// TwinCAT 3 PLC project Untitled1
// ProgramVersion: 3.1.4023.0
// libraries:
//   Tc2_Standard, * (Beckhoff Automation GmbH)
//   Tc2_System, * (Beckhoff Automation GmbH)
//   Tc2_Utilities, * (Beckhoff Automation GmbH)
//   Tc3_Database, * (Beckhoff Automation GmbH)
//   Tc3_Module, * (Beckhoff Automation GmbH)
// project tree:
//   DUTs/ ExcelInfo.TcDUT, ST_AccessConnectionInfo.TcDUT, ST_datastruct.TcDUT, st_DBInfo.TcDUT, st_InsertData.TcDUT (not stored), ST_mongoDBConnectionInfo.TcDUT, ST_MYSQLConnectionInfo.TcDUT, ST_ReturnBetweenDates.TcDUT, ST_ReturnedData_mysql_access.TcDUT, ST_SQLiteConnectionInfo.TcDUT, test.TcDUT
//   / PlcTask.TcTTO
//   POUs/ fb_ConnectDB.TcPOU, fb_CreateTable.TcPOU, fb_DBSRVCreateTable.TcPOU, fb_datareturn.TcPOU, fb_DBSRVdatareturn.TcPOU, fb_DBWrite.TcPOU, fb_DBSRVInsertRecord.TcPOU, MAIN.TcPOU

CONFIGURATION Untitled1
    RESOURCE PLC ON TwinCAT3
        TASK PlcTask(INTERVAL := T#1ms, PRIORITY := 20);
        PROGRAM MAIN WITH PlcTask : MAIN;
    END_RESOURCE
END_CONFIGURATION

// ---- DUTs/ExcelInfo.TcDUT
TYPE ExcelInfo :
STRUCT
	ColumnName:STRING(50):='';
	ColumnNumber:INT:=0;
	bready:BOOL:=FALSE;
	path:STRING(200):='';
END_STRUCT
END_TYPE

// ---- DUTs/ST_AccessConnectionInfo.TcDUT
TYPE ST_AccessConnectionInfo :
STRUCT
	Path:STRING(255);
END_STRUCT
END_TYPE

// ---- DUTs/ST_datastruct.TcDUT
TYPE ST_datastruct :
STRUCT
	//datum:DATE;
	temp_set:DINT:=0;
	temp_act:DINT:=0;
	hum_set:DINT:=0;
	hum_act:DINT:=0;
	further_parameter1:DINT:=0;
END_STRUCT
END_TYPE

// ---- DUTs/st_DBInfo.TcDUT
TYPE st_DBInfo :
STRUCT
	AccessConnectionInfo:ST_AccessConnectionInfo;
	DBMS:STRING(50):='';
	//table:STRING(50);
	MYSQLConnectionInfo:ST_MYSQLConnectionInfo;
	MongoDBConnectionInfo:ST_MongoDBConnectionInfo;
	SQLiteConnectionInfo:ST_SQLiteConnectionInfo;
END_STRUCT
END_TYPE

// ---- DUTs/ST_mongoDBConnectionInfo.TcDUT
TYPE ST_mongoDBConnectionInfo :
STRUCT
	MongoDBDatabase:STRING(50):='';
	
END_STRUCT
END_TYPE

// ---- DUTs/ST_MYSQLConnectionInfo.TcDUT
TYPE ST_MYSQLConnectionInfo :
STRUCT
	user:STRING(50):='';
	password:STRING(100):='';
	server:STRING(100):='localhost';
	DB:String(50):='';
END_STRUCT
END_TYPE

// ---- DUTs/ST_ReturnBetweenDates.TcDUT
TYPE ST_ReturnBetweenDates :
STRUCT
	kezdo : STRING;
	veg:STRING;
	table:STRING(50);
	//bExecute:BOOL:=FALSE;
	//DBMS: STRING(50);
	
END_STRUCT
END_TYPE

// ---- DUTs/ST_ReturnedData_mysql_access.TcDUT
TYPE ST_ReturnedData_mysql_access :
STRUCT
	Datum:DATE_AND_TIME;
	temp_set:DINT;
	temp_act:DINT;
	hum_set:dINT;
	hum_act:DINT;
END_STRUCT
END_TYPE

// ---- DUTs/ST_SQLiteConnectionInfo.TcDUT
TYPE ST_SQLiteConnectionInfo :
STRUCT
	Path:STRING(255);
END_STRUCT
END_TYPE

// ---- DUTs/test.TcDUT
TYPE test :
STRUCT
	dbName:STRING(50);
	dbID:UINT;
	dbtable:STRING(50);
	excelColName:STRING(50);
	excelcol:INT;
	connector:STRING(50);
	
END_STRUCT
END_TYPE

// ---- POUs/MAIN.TcPOU
PROGRAM MAIN
VAR
	//dbserver
	DBSRVdatareturn:fb_DBSRVdatareturn;
	
	st_insertData:st_insertData;
	st_returneddata:ST_ReturnedData_mysql_access;
	//csharp
	DataReturn:fb_datareturn;
	ConnectDB:fb_ConnectDB;
	DBWrite:fb_DBWrite;
	Createtable:fb_CreateTable;
	//időmérés
	bStart:BOOL:=FALSE;
	TONTimer:TON;
	falling_trig:F_TRIG;
	time1:TIME;
	time_array: ARRAY [1..80] OF TIME;
	timearraylenght:INT:=80;
	counter:INT:=1;
	
	nstep:INT:=10;
	testarray: ARRAY[1..21] OF test;
	testarrayLenght:INT:=21;
	i:INT:=1;
	ExcelInfo:Excelinfo;
	
	startprocess: NT_startprocess;
	startprocessExcel:ARRAY [1..21] OF NT_startprocess;
END_VAR

CASE nstep OF 
	5://idle
		
	10://init
		connectdb.DBInfo.MYSQLConnectionInfo.DB:='speedTest';
		connectdb.DBInfo.MYSQLConnectionInfo.password:='132435465768';
		connectdb.DBInfo.MYSQLConnectionInfo.server:='localhost';
		connectdb.DBInfo.MYSQLConnectionInfo.user:='root';
		
		connectdb.DBInfo.SQLiteConnectionInfo.Path:='D:\Egyetemes szarok 6. félév\PLC projekt\speedTest.db';
		
		connectdb.DBInfo.MongoDBConnectionInfo.MongoDBDatabase:='speedTest';
		
		connectdb.DBInfo.AccessConnectionInfo.Path:='D:\Egyetemes szarok 6. félév\PLC projekt\speedTest.accdb';
		
		testarray[1].connector:='dbserver';
		testarray[1].dbID:=1;
		testarray[1].dbtable:='10_record';
		testarray[1].excelColName:='access 10 rec plc';
		testarray[1].excelcol:=1;
		
		testarray[2].connector:='dbserver';
		testarray[2].dbID:=1;
		testarray[2].dbtable:='100_record';
		testarray[2].excelColName:='access 100 rec plc';
		testarray[2].excelcol:=3;
		
		testarray[3].connector:='dbserver';
		testarray[3].dbID:=1;
		testarray[3].dbtable:='1000_record';
		testarray[3].excelColName:='access 1000 rec plc';
		testarray[3].excelcol:=5;
		
		testarray[4].connector:='csharp';
		testarray[4].dbName:='SQLite';
		testarray[4].dbtable:='10_record';
		testarray[4].excelColName:='sqlite 100 rec csarp';
		testarray[4].excelcol:=7;
		
		testarray[5].connector:='csharp';
		testarray[5].dbName:='MySQL';
		testarray[5].dbtable:='10_record';
		testarray[5].excelColName:='MYsql 10 rec csharp';
		testarray[5].excelcol:=9;
		
		testarray[6].connector:='csharp';
		testarray[6].dbName:='SQLite';
		testarray[6].dbtable:='100_record';
		testarray[6].excelColName:='sqlite 100 rec csarp';
		testarray[6].excelcol:=11;
		
		testarray[7].connector:='csharp';
		testarray[7].dbName:='MySQL';
		testarray[7].dbtable:='100_record';
		testarray[7].excelColName:='MYsql 100 rec csharp';
		testarray[7].excelcol:=13;
		
		testarray[8].connector:='csharp';
		testarray[8].dbName:='SQLite';
		testarray[8].dbtable:='1000_record';
		testarray[8].excelColName:='sqlite 1000 rec csarp';
		testarray[8].excelcol:=15;
		
		
		testarray[9].connector:='csharp';
		testarray[9].dbName:='MySQL';
		testarray[9].dbtable:='1000_record';
		testarray[9].excelColName:='MYsql 1000 rec csharp';
		testarray[9].excelcol:=17;
		
		testarray[10].connector:='csharp';
		testarray[10].dbName:='Access';
		testarray[10].dbtable:='10_record';
		testarray[10].excelColName:='Access 10 rec csharp';
		testarray[10].excelcol:=19;
		
		testarray[11].connector:='csharp';
		testarray[11].dbName:='Access';
		testarray[11].dbtable:='100_record';
		testarray[11].excelColName:='Access 100 rec csharp';
		testarray[11].excelcol:=21;
		
		testarray[12].connector:='csharp';
		testarray[12].dbName:='Access';
		testarray[12].dbtable:='1000_record';
		testarray[12].excelColName:='Access 1000 rec csharp';
		testarray[12].excelcol:=23;
		
		testarray[13].connector:='csharp';
		testarray[13].dbName:='MongoDB';
		testarray[13].dbtable:='10_record';
		testarray[13].excelColName:='MongoDB 10 rec csharp';
		testarray[13].excelcol:=25;
		
		testarray[14].connector:='csharp';
		testarray[14].dbName:='MongoDB';
		testarray[14].dbtable:='100_record';
		testarray[14].excelColName:='MongoDB 100 rec csharp';
		testarray[14].excelcol:=27;
		
		testarray[15].connector:='csharp';
		testarray[15].dbName:='MongoDB';
		testarray[15].dbtable:='1000_record';
		testarray[15].excelColName:='MongoDB 1000 rec csharp';
		testarray[15].excelcol:=29;
		
		testarray[16].connector:='dbserver';
		testarray[16].dbID:=2;
		testarray[16].dbtable:='10_record';
		testarray[16].excelColName:='MySQL 10 rec DBserver';
		testarray[16].excelcol:=31;
		
		testarray[17].connector:='dbserver';
		testarray[17].dbID:=2;
		testarray[17].dbtable:='100_record';
		testarray[17].excelColName:='MySQL 100 rec DBserver';
		testarray[17].excelcol:=33;
		
		testarray[18].connector:='dbserver';
		testarray[18].dbID:=2;
		testarray[18].dbtable:='1000_record';
		testarray[18].excelColName:='MySQL 1000 rec DBserver';
		testarray[18].excelcol:=35;
		
		testarray[19].connector:='dbserver';
		testarray[19].dbID:=3;
		testarray[19].dbtable:='$'10_record$'';
		testarray[19].excelColName:='SQLite 10 rec DBserver';
		testarray[19].excelcol:=37;
		
		testarray[20].connector:='dbserver';
		testarray[20].dbID:=3;
		testarray[20].dbtable:='$'100_record$'';
		testarray[20].excelColName:='SQLite 100 rec DBserver';
		testarray[20].excelcol:=39;
		
		testarray[21].connector:='dbserver';
		testarray[21].dbID:=3;
		testarray[21].dbtable:='$'1000_record$'';
		testarray[21].excelColName:='SQLite 1000 rec DBserver';
		testarray[21].excelcol:=41;
		
		//testarray[16].connector:='csharp';
		//testarray[16].dbName:='MongoDB';
		//testarray[16].dbtable:='10000_record';
		//testarray[16].excelColName:='MongoDB 10000 rec csharp';
		//testarray[16].excelcol:=16;
		
		startprocess(NETID:='',
					PATHSTR:='D:\Egyetemes szarok 6. félév\PLC projekt\final with entity V2\bin\Debug\final with entity.exe',
					DIRNAME:='D:\Egyetemes szarok 6. félév\PLC projekt\final with entity V2\bin\Debug',
					Comndline:='start final with entity.exe',//'win.ini',
					START:=TRUE,
					tMOUT:=T#5S);
					IF NOT startprocess.BUSY THEN
						nstep:=20;   
					END_IF
		
		
	20:	// choose connector
		IF testarray[i].connector='csharp' THEN
			nstep:=30;
		END_IF
		IF testarray[i].connector='dbserver' THEN
			nstep:=100;
		END_IF
		
	30://c# MEGOLDÁS
		//connect 
		//start timer	
		
		tontimer.IN:=TRUE;
		connectdb.DBInfo.DBMS:=testarray[i].dbName;
		connectdb.connect();
		IF ConnectDB.bConnected THEN
				nstep:=40;
		END_IF
	40://lekérdezés	
		DataReturn.ReturnBetweenDates.kezdo:='2020-07-01 12:00:00';
			DataReturn.ReturnBetweenDates.veg:='2020-08-30 12:00:00';
			Datareturn.ReturnBetweenDates.table:=testarray[i].dbtable;//'1000_record';
			//IF NOT datareturn.bExecute THEN
				Datareturn.execute();
			//END_IF
			nstep:=50;
			
		//	IF DataReturn.bReady THEN
				 //
				// Connectdb.disconnect();
				
				//stop timer
			//	tontimer.IN:=FALSE;
				//nstep:=30;
			//END_IF
	50: 
		IF DataReturn.bReady THEN
				 //
				 
				 Connectdb.disconnect();
				IF NOT connectdb.bConnected THEN
					tontimer.IN:=FALSE;
					datareturn.reset();
					nstep:=30;
				END_IF
				//stop timer
				
			END_IF
		
		100:// db server megoldás
			tontimer.IN:=TRUE;
			IF testarray[i].dbID=1 THEN
				DBSRVdatareturn.start:= '#7/1/2020 12:0:0#';
				DBSRVdatareturn.end:=' #8/30/2020 15:0:0#';
			ELSE 
				DBSRVdatareturn.start:='$'2020-07-01 15:00:01$'' ;
				DBSRVdatareturn.end:= '$'2020-08-30 15:00:01$'';	
			END_IF
			
			DBSRVdatareturn(DBID:=testarray[i].dbID,
				//table:='$'10_record$'',
				table:=testarray[i].dbtable,
				bExecute:=TRUE);
				
				//kezdo:='$'2020-07-01 15:00:01$'',
				//veg:='$'2020-08-30 15:00:01$''); //// a dátumok szintén aposztrófok közzé mennek
			IF DBSRVdatareturn.bReady THEN
				DBSRVdatareturn.Reset();
				DBSRVdatareturn.ClearArray();
				tontimer.IN:=FALSE;
				
			END_IF
			
		200: // write to excel
			ExcelInfo.ColumnName:=testarray[i].excelColName;
				ExcelInfo.ColumnNumber:=testarray[i].excelcol;
				excelinfo.path:='D:\Egyetemes szarok 6. félév\PLC projekt\Adatkiértékelés.xlsx';
				startprocessExcel[i](NETID:='',
							PATHSTR:='D:\Egyetemes szarok 6. félév\PLC projekt\Twincat array to excel\obj\Debug\Twincat array to excel.exe',
							DIRNAME:='D:\Egyetemes szarok 6. félév\PLC projekt\Twincat array to excel\obj\Debug',
							Comndline:='start Twincat array to excel.exe',
							START:=TRUE,
							tMOUT:=T#5S);
				IF NOT startprocessExcel[i].BUSY AND excelinfo.bready THEN
					IF i<=testarrayLenght THEN
						i:=i+1;
					ELSE
						nstep:=	5;
					END_IF
					
					excelinfo.bready:=FALSE;
					//startprocessExcel[i].START:=FALSE;
					nstep:=20;
				END_IF				
END_CASE
	
falling_trig(clk:=tontimer.IN);
	IF falling_trig.Q THEN
		time1:=tontimer.ET;
		IF counter<timearraylenght+1 THEN
			time_array[counter]:=time1;
			counter:=counter+1;
			tontimer.IN:=FALSE;
			
		ELSE
			counter:=1;	
			nstep:=200;
			
		END_IF
	END_IF
	tontimer(PT:=T#60S);

END_PROGRAM

// ---- POUs/fb_DBSRVdatareturn.TcPOU
FUNCTION_BLOCK fb_DBSRVdatareturn
VAR_INPUT
	dbid:UINT;
	table:STRING(50);
	start:STRING(100);
	end:STRING(100);
	bExecute:BOOL;
	
	
END_VAR
VAR_OUTPUT
	ReadStruct: ARRAY [0..1001] OF ST_ReturnedData_mysql_access;
	
	bReady:BOOL:=FALSE;
	Error:BOOL:=FALSE;
END_VAR
VAR
	sCmd:STRING(255):='';
	nstep:int:=10;
	SQLresult: FB_SQLResultEvt(sNetID:='', tTimeout:=T#5S);
	SQLcommand: FB_SQLCommandEvt(sNetid:='',tTimeout:=T#5S);
	Connectdb: FB_sqldatabaseevt(SNetID:='', tTimeout:=T#5S);
	//bExecute:BOOL:=FALSE;
	connected:BOOL:=FALSE;
	
END_VAR

	
		
IF bExecute THEN
	CASE nstep OF
	10:
				sCmd:=CONCAT('SELECT Dátum, temp_set, temp_act, hum_set, hum_act FROM ',table);
				sCmd:=concat(sCmd, ' WHERE Dátum BETWEEN ');
				sCmd:=concat(sCmd , start);
				sCmd:=Concat(sCmd , ' AND ');
				sCmd:=concat(sCmd , end);
				sCmd:=concat(sCmd,';');
				nstep:=20;
	20:		IF connectDB.Connect(dbid) THEN
				IF connectdb.bError THEN
					Error:=TRUE;
				ELSE
					connected:=TRUE;
				END_IF
			END_IF
			IF connected AND NOT connectDB.bBusy THEN 
				IF connectDB.CreateCmd(pSQLCommand:= ADR(SQLcommand)) THEN
					nstep:=30;
				END_IF
			END_IF	
			
						
	30:
			IF SQLcommand.ExecuteDataReturn(pSQLCmd:=ADR(sCmd),
										cbSQLCmd:=SIZEOF(sCmd),
										pSQLDBResult:=ADR(SQLResult))
			THEN
			IF sqlcommand.bError THEN
				Error:=TRUE;
			ELSE
			IF NOT SQLcommand.bBusy THEN
				nstep:=40;
			END_IF
			END_IF
			END_IF
	40:	IF SQLResult.Read(nStartindex:= 1,
						  nRecordCount:=1001,
						  pData:=ADR(ReadStruct),
						  cbData:=SIZEOF(ReadStruct),
							TRUE, TRUE)
		THEN
		IF sqlresult.bError THEN
			Error:=TRUE;
		ELSE
		IF NOT SQLResult.bBusy	THEN
			nstep:=50;
			
		END_IF
		END_IF
		END_IF	
	50:
		IF connectDB.Disconnect() THEN
			IF connectdb.bError THEN
				Error:=TRUE;
			ELSE
				connected:=FALSE;
				bReady:=TRUE;
				bExecute:=FALSE;	
		END_IF
		END_IF	
END_CASE
END_IF

METHOD ClearArray : BOOL
VAR_INPUT
END_VAR
memset(adr(readstruct),0,sizeof(readstruct));
END_METHOD

METHOD Reset : BOOL
VAR_INPUT
END_VAR
bReady:=FALSE;
nstep:=10;
END_METHOD

END_FUNCTION_BLOCK

// ---- POUs/fb_datareturn.TcPOU
FUNCTION_BLOCK fb_datareturn
VAR_INPUT
	
	ReturnBetweenDates:ST_ReturnBetweenDates;
END_VAR

VAR_OUTPUT
	recordarray: ARRAY [0..1500] OF STRING(100);
	bReady:bool:=false;
END_VAR
VAR
	bExecute:BOOL:=FALSE;
	i:int;
	
END_VAR

METHOD ClearRecordArray : BOOL
VAR_INPUT
END_VAR
i:=0;
FOR i:=0 TO 1500 BY 1 DO
	RecordArray[i]:='';
END_FOR
END_METHOD

METHOD execute : BOOL
VAR_INPUT
END_VAR
bExecute:=TRUE;
END_METHOD

METHOD reset : BOOL
VAR_INPUT
END_VAR
bExecute:=FALSE;


bReady:=false;
END_METHOD

END_FUNCTION_BLOCK

// ---- POUs/fb_ConnectDB.TcPOU
FUNCTION_BLOCK fb_ConnectDB
VAR_INPUT
	DBInfo:st_DBInfo;
	bConnect:BOOL:=FALSE;
	
END_VAR
VAR_OUTPUT
	bConnected:BOOL:=FALSE;
END_VAR
VAR
END_VAR

METHOD connect : BOOL
VAR_INPUT
END_VAR
bConnect:=true;
END_METHOD

METHOD disconnect : BOOL
VAR_INPUT
END_VAR
bConnect:=false;
END_METHOD

END_FUNCTION_BLOCK

// ---- POUs/fb_DBWrite.TcPOU
FUNCTION_BLOCK fb_DBWrite
VAR_INPUT
	DataStruct:ST_DataStruct;
	Table:String(50);
END_VAR
VAR_OUTPUT
	bReady:bool:=false;
END_VAR
VAR
	bExecute:BOOL:=FALSE;
	
END_VAR

METHOD execute : BOOL
VAR_INPUT
END_VAR
bExecute:=TRUE;
END_METHOD

METHOD reset : BOOL
VAR_INPUT
END_VAR
bExecute:=FALSE;
bReady:=false;
END_METHOD

END_FUNCTION_BLOCK

// ---- POUs/fb_CreateTable.TcPOU
FUNCTION_BLOCK fb_CreateTable
VAR_INPUT
	tablename:STRING(50);
END_VAR
VAR_OUTPUT
	bReady:BOOL:=FALSE;
END_VAR
VAR
	bExecute:Bool:=false;
END_VAR

METHOD execute : BOOL
VAR_INPUT
END_VAR
bExecute:=TRUE;
END_METHOD

METHOD reset : BOOL
VAR_INPUT
END_VAR
bExecute:=FALSE;
bReady:=false;
END_METHOD

END_FUNCTION_BLOCK

// ---- POUs/fb_DBSRVCreateTable.TcPOU
FUNCTION_BLOCK fb_DBSRVCreateTable
VAR_INPUT
	table:STRING(50);
	bExecute:BOOL;
	DBID:UINT;
	
END_VAR
VAR_OUTPUT
	bError:BOOL:=FALSE;
	bReady:BOOL:=FALSE;
END_VAR
VAR
	sCmd:STRING(255);
	nstep:INT:=10;
	SQLcommand: FB_SQLCommandEvt(sNetid:='',tTimeout:=T#5S);
	Connectdb: FB_sqldatabaseevt(SNetID:='', tTimeout:=T#5S);
	connected:BOOL:=FALSE;
END_VAR

IF bExecute THEN
CASE nstep OF
	10:
		IF connectDB.Connect(DBID) THEN
			
			IF connectdb.bError THEN
				bError:=TRUE;
			ELSE
				connected:=TRUE;	
			END_IF
		END_IF
		IF connected and NOT connectDB.bBusy THEN 
			IF connectDB.CreateCmd(pSQLCommand:= ADR(SQLcommand)) THEN
				nstep:=20;
			END_IF
		END_IF
	20:	
	
		sCmd:=concat('CREATE TABLE ', table);
		sCmd:=concat(sCmd,'(Dátum DATETIME ,
  						temp_set INTEGER ,
  						temp_act INTEGER ,
  						hum_set INTEGER ,
 						 hum_act INTEGER );');
		nstep:=30;
		
	30:
		IF SQLcommand.Execute(pSQLCmd:=ADR(sCmd),
							cbSQLCmd:=SIZEOF(sCmd))
		THEN
			IF sqlcommand.bError THEN
				berror:=TRUE;
			ELSE
			IF NOT SQLcommand.bBusy THEN
				nstep:=40;
			
			END_IF
			END_IF
		END_IF
	40:	
		IF connectDB.Disconnect() THEN
			IF connectdb.bError THEN
				bError:=TRUE;
			ELSE
				connected:=FALSE;
			bReady:=TRUE;
			bExecute:=FALSE;	
		END_IF
		END_IF	
			
END_CASE
END_IF

METHOD Reset : BOOL
VAR_INPUT
END_VAR
bReady:=FALSE;
nstep:=10;
END_METHOD

END_FUNCTION_BLOCK

// ---- POUs/fb_DBSRVInsertRecord.TcPOU
FUNCTION_BLOCK fb_DBSRVInsertRecord
VAR_INPUT
	InsertData:ST_InsertData;
	table:STRING(50);
	DBID:UINT;
	bExecute:bool;
	
END_VAR
VAR_OUTPUT
	bError:BOOL:=FALSE;
	bReady:BOOL:=FALSE;
	
END_VAR
VAR
	nstep:INT:=10;
	sCmd:STRING(255);
	SQLcommand: FB_SQLCommandEvt(sNetid:='',tTimeout:=T#5S);
	Connectdb: FB_sqldatabaseevt(SNetID:='', tTimeout:=T#5S);
	connected:BOOL:=FALSE;
	
END_VAR

IF bExecute THEN
CASE nstep OF 
	10:
			sCmd:=concat('insert into ',table);
			sCmd:=concat(sCmd,  ' (Dátum , temp_set, temp_act, hum_set, hum_act ) values ('); //{Datum},{temp_set},{temp_act},{hum_set}, {hum_act})');
			sCmd:=concat(sCmd,insertdata.Datum);
			sCmd:=concat(sCmd,', ');
			sCmd:=concat(sCmd,insertdata.temp_set);
			sCmd:=concat(sCmd,', ');
			sCmd:=concat(sCmd,insertdata.temp_act);
			sCmd:=concat(sCmd,', ');
			sCmd:=concat(sCmd, insertdata.hum_set);
			sCmd:=concat(sCmd,', ');
			sCmd:=concat(sCmd,insertdata.hum_act);
			sCmd:=concat(sCmd,')');
			nstep:=20;
	20:
			IF connectDB.Connect(DBID) THEN
				IF connectdb.bError THEN
					bError:=TRUE;
				ELSE
					connected:=TRUE;	
				END_IF
			END_IF
			IF connected AND NOT connectDB.bBusy THEN 
				IF connectDB.CreateCmd(pSQLCommand:= ADR(SQLcommand)) THEN
					nstep:=30;
				END_IF
			END_IF		
	30:
		IF SQLcommand.Execute(pSQLCmd:=ADR(sCmd),
							cbSQLCmd:=SIZEOF(sCmd))
			THEN
			IF sqlcommand.bError THEN
				Berror:=TRUE;
			ELSE
			IF NOT SQLcommand.bBusy THEN
				nstep:=40;
			END_IF
			END_IF
		END_IF
	40:	
		IF connectDB.Disconnect() THEN
			IF connectdb.bError THEN
				bError:=TRUE;
			ELSE
				connected:=FALSE;
				bReady:=TRUE;
				bExecute:=FALSE;	
		END_IF
		END_IF		
		
END_CASE
END_IF

METHOD Reset : BOOL
VAR_INPUT
END_VAR
bReady:=FALSE;
nstep:=10;
END_METHOD

END_FUNCTION_BLOCK
